{attribute 'GeneratedUsingTerminal: EL1258-0000-0016'}
{attribute addProperty BoxType "EL1258-0000-0016"}
{attribute addProperty Id "No_of_input_eventsUSINT1Input_stateBOOL1Input_buffer_overflowBOOL1Input_cycle_counterBYTE1Events_in_input_bufferUSINT1Input_order_feedbackUSINT1"}
{attribute addProperty CRC "1454809052"}
{attribute addProperty Size "6"}
TYPE Status_56B69FDC :
STRUCT
	{attribute addProperty Name "No_of_input_events"}
	No_of_input_events : USINT;
	{attribute addProperty Name "Input_state"}
	Input_state : BOOL;
	{attribute addProperty Name "Input_buffer_overflow"}
	Input_buffer_overflow : BOOL;
	{attribute addProperty Name "Input_cycle_counter"}
	Input_cycle_counter : BYTE;
	{attribute addProperty Name "Events_in_input_buffer"}
	Events_in_input_buffer : USINT;
	{attribute addProperty Name "Input_order_feedback"}
	Input_order_feedback : USINT;
END_STRUCT
END_TYPE

(* stored: Version 1.2.0.0, ProductVersion 3.1.4024.9
   DUT Status_56B69FDC: Id {7031898b-ea98-44fa-89eb-47935ad1f413} *)
